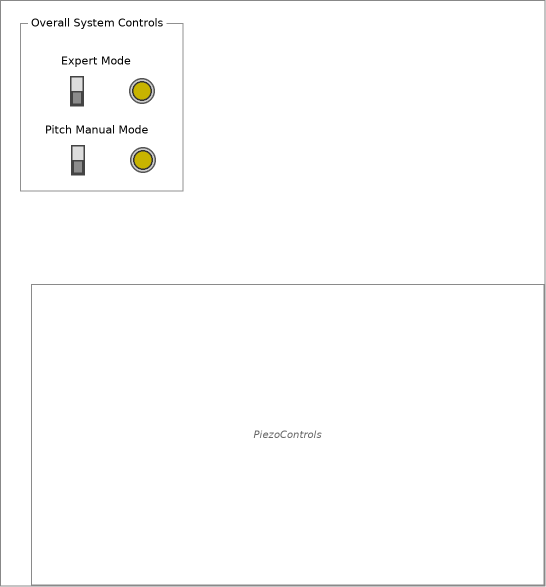
VISUALIZATION Visualization  // 546x587
    GroupBox (20,15 163x176), "Overall System Controls"
        DipSwitch (17,61 80x30), tooltip "Puts the pitch control function block into manual mode. In manual mode the piezo and stepper movements are completely independent of one another and no coordinated actions take place. Limit switches are still respected.", variable: MAIN.ExpertMode, behaviour: TOGGLE, style: Switch-DipSwitch-Gray
        Label (20,31 112x30), "Expert Mode"
        Lamp1 (107,61 30x30), variable: MAIN.ExpertMode, style: Lamp-Lamp1-Yellow
        DipSwitch (18,130 80x30), tooltip "Puts the pitch control function block into manual mode. In manual mode the piezo and stepper movements are completely independent of one another and no coordinated actions take place. Limit switches are still respected.", variable: MAIN.DirectPiezoMode, behaviour: TOGGLE, style: Switch-DipSwitch-Gray
        Label (21,100 112x30), "Pitch Manual Mode"
        Lamp1 (108,130 30x30), variable: MAIN.PitchControl.DirectPiezoControl, style: Lamp-Lamp1-Yellow
    Frame (31,284 513x301)
        shows PiezoControls(Piezo := HOMS1_Pitch.Piezo, ActPos := HOMS1_Pitch.Stepper)
END_VISUALIZATION

(* stored: Version 1.1.0.1, ProductVersion 3.1.4020.12
   Visu Visualization: Id {2842b111-ef8a-453c-b858-3dcb33a12eaf} *)
